FUNCTION_BLOCK SystemFunktionen
VAR_INPUT
END_VAR
VAR_OUTPUT
END_VAR
VAR
	Timer_1Hz: TON;	
	Timer_1_25Hz: TON;
END_VAR

Timer_1Hz(IN:= NOT Timer_1Hz.Q, PT:= T#1S);
Blinker.Clock_1Hz := Timer_1Hz.ET < T#500MS;

Timer_1_25Hz(IN:= NOT Timer_1_25Hz.Q, PT:= T#800MS);
Blinker.Clock_1_25Hz:= Timer_1_25Hz.ET < T#400MS;

END_FUNCTION_BLOCK

(* stored: Version 1.1.0.1, ProductVersion 3.1.4024.5
   POU SystemFunktionen: Id {21a6b941-b515-4a59-93af-71953637eed8}, SpecialFunc None *)
